	ElCurrentL3Base			: ARRAY[1..2] OF ARRAY[1..100] OF REAL := 
								[
								[0, 0, 0.1, 0.3, 0.45, 0.60, 0.70, 0.80, 0.95, 1.1, 1.3, 1.4, 1.55, 1.6, 1.59,1.55, 
								1.45, 1.3, 1.2, 1.1, 1.05, 1.0, 0.95, 0.9, 0.85, 0.83, 0.80, 0.78, 0.75, 0.74, 0.72,
								0.70, 0.69, 0.69, 0.69, 0.68, 0.68, 0.67, 0.67, 0.65, 0.64, 0.62, 0.60, 0.58, 0.58, 0.57, 0.56, 0.55, 0.55,
								0, 0, 0, 0, 0, 0, 0, 0, 0, 0],
								[0, 0, 0.1, 0.2, 0.3, 0.55, 1.0, 1.3, 1.5, 1.7, 1.8, 1.81, 1.7, 1.5, 1.2, 1.22, 1.19, 1.23,
								1.19, 1.21, 1.18, 1.22, 1.19, 1.23, 1.17, 1.21, 1.20, 1.18, 1.21, 1.18, 1.22, 1.17, 1.23,
								1.19, 1.21, 1.19, 1.20, 1.19, 1.20, 1.19, 1.21, 1.20, 1.20, 1.22, 1.19, 1.21, 1.18, 1.21, 1.2, 1.2,
								1.21, 1.20, 1.20, 1.22, 1.19, 1.21, 1.18, 1.21, 1.2, 1.2]];
END_VAR

IF GVL_Visu.ButtonStart THEN
	
	GVL_Visu.LineRunning := TRUE;
	// simulate motor running signals
	tp1Motor[1](IN:= NOT tp2Motor[1].Q, PT:= T#1S);
	tp2Motor[1](IN:= NOT tp1Motor[1].Q, PT:= T#500MS);
	
	tp1Motor[2](IN:= NOT tp2Motor[2].Q, PT:= T#2S);
	tp2Motor[2](IN:= NOT tp1Motor[2].Q, PT:= T#300MS);
	
	tp1Motor[3](IN:= NOT tp2Motor[3].Q, PT:= T#1.7S);
	tp2Motor[3](IN:= NOT tp1Motor[3].Q, PT:= T#500MS);
	
	tp1Motor[4](IN:= NOT tp2Motor[4].Q, PT:= T#1S);
	tp2Motor[4](IN:= NOT tp1Motor[4].Q, PT:= T#1S);
	
	tp1Motor[5](IN:= NOT tp2Motor[5].Q, PT:= T#500MS);
	tp2Motor[5](IN:= NOT tp1Motor[5].Q, PT:= T#2S);
	
	tp1Motor[6](IN:= NOT tp2Motor[6].Q, PT:= T#1S);
	tp2Motor[6](IN:= NOT tp1Motor[6].Q, PT:= T#300MS);
	
	// simulate auto/manual mode
	tp1AutoMode(IN:= NOT tp2AutoMode.Q, PT:= tp1AutoModeTime);
	tp2AutoMode(IN:= NOT tp1AutoMode.Q, PT:= tp2AutoModeTime);
	
	rtrigAutoMode(CLK:=tp1AutoMode.Q);
	
	// generate random time windows of auto and manual period  
	IF  rtrigAutoMode.Q THEN
		rndTime1 := RDM2(last:=2, low:=0, high:=70);
		tp1AutoModeTime:=T#5S + INT_TO_TIME(rndTime1*100);
		
		rndTime2 := RDM2(last:=5, low:=0, high:=30);
		tp2AutoModeTime:=T#2S + INT_TO_TIME(rndTime2*100);
	END_IF

	GVL_Visu.AutoMode := tp2AutoMode.Q;
	
	
	// simulate vibration sensors
	FOR idx := 1 TO 6 DO
		GVL_Visu.MotorRunning[idx] := tp1Motor[idx].Q;
		
		GVL_Visu.VibrationSensorX[idx] := VibSensorBase[idx] + RDM(0.4);
		GVL_Visu.VibrationSensorY[idx] := VibSensorBase[idx] + RDM(0.2);
		GVL_Visu.VibrationSensorZ[idx] := VibSensorBase[idx] + RDM(0.8);	
	END_FOR
	
	// simulate air supply sensors
	GVL_Visu.AirFlowRate 		:= AirFlowRateBase + 2* RDM(0.5);
	GVL_Visu.AirPressure		:= AirPressureBase + 2 * RDM(0.9); 
	GVL_Visu.AirTemperature		:= AirTemperatureBase + RDM(0.3);
	
	// simulate air valves
	AirValve[1](StartSim			:= TRUE, 
			    ExtendCmdTime		:= T#500MS,
			    ExtendTime 			:= T#1800MS,
			    RetractCmdTime 		:= T#600MS,
			    RetractTime  		:= T#2000MS);
			  
	AirValve[2](StartSim			:= TRUE, 
			    ExtendCmdTime		:= T#50MS,
			    ExtendTime 			:= T#180MS,
			    RetractCmdTime 		:= T#50MS,
			    RetractTime  		:= T#145MS);
				
	AirValve[3](StartSim			:= TRUE, 
			    ExtendCmdTime		:= T#100MS,
			    ExtendTime 			:= T#1200MS,
			    RetractCmdTime 		:= T#120MS,
			    RetractTime  		:= T#1500MS);
				
	AirValve[4](StartSim			:= TRUE, 
			    ExtendCmdTime		:= T#30MS,
			    ExtendTime 			:= T#120MS,
			    RetractCmdTime 		:= T#30MS,
			    RetractTime  		:= T#120MS);
				
	FOR idx := 1 TO 4 DO
		GVL_Visu.AirValve[idx].ExtendCmd := AirValve[idx].ExtendCmd;
		GVL_Visu.AirValve[idx].ExtendFeedback := AirValve[idx].ExtendFeedback;
		GVL_Visu.AirValve[idx].RetractCmd := AirValve[idx].RetractCmd;
		GVL_Visu.AirValve[idx].RetractFeedback := AirValve[idx].RetractFeedback;
		GVL_Visu.AirValvePositionSim[idx] := SEL (NOT GVL_Visu.AirValveEnable[idx], AirValve[idx].nState, 0);
	END_FOR
	
	// simulate product position on the conveyor
	tonProductPos(IN:= NOT tonProductPos.Q, PT:=T#200MS);
	IF tonProductPos.Q THEN
		GVL_Visu.ProductPosition := GVL_Visu.ProductPosition + TO_INT(GVL_Visu.LineSpeed / 5);
	END_IF
	
	IF GVL_Visu.ProductPosition >= 190 THEN
		GVL_Visu.ProductPosition := 0;
	END_IF
	
	// simulate product sensor acitivation
	IF GVL_Visu.ProductPosition >= 175 AND
		 GVL_Visu.ProductPosition <190 THEN
	GVL_Visu.SensorProductActive := TRUE;
	ELSE
		GVL_Visu.SensorProductActive := FALSE;
	END_IF;
	
	// simulate product counting
	rtrigProductSensor(CLK:=GVL_Visu.SensorProductActive);
	IF rtrigProductSensor.Q THEN
		GVL_Visu.OkProductCount := GVL_Visu.OkProductCount + 1;
	END_IF
	
	// simulate electrical current curve of motor 1
	IF GVL_Visu.MotorRunning[1] THEN
		ElecSample1 := ElecSample1+1;
		ElecSample1 := SEL(ElecSample1=60, ElecSample1, 1);
		IF ElecSample1 < 20 OR ElecSample1 > 40 THEN
			ElecCurrentOffsetL1 := RDM(0.67) * 0.05;
			ElecCurrentOffsetL2 := RDM(0.23) * 0.05;
			ElecCurrentOffsetL3 := RDM(0.72) * 0.05;
		ELSE
			ElecCurrentOffsetL1 := RDM(0.31) * 0.05;
			ElecCurrentOffsetL2 := RDM(0.63) * 0.05;
			ElecCurrentOffsetL3 := RDM(0.46) * 0.05;
		END_IF
		GVL_Visu.ElCurrentL1[1] := 	ElCurrentL1Base[1][ElecSample1] + ElecCurrentOffsetL1;
		GVL_Visu.ElCurrentL2[1] := 	ElCurrentL2Base[1][ElecSample1] + ElecCurrentOffsetL2;
		GVL_Visu.ElCurrentL3[1] := 	ElCurrentL3Base[1][ElecSample1] + ElecCurrentOffsetL3;
	ELSE
		ElecSample1 := 0;
		GVL_Visu.ElCurrentL1[1] := 0;
		GVL_Visu.ElCurrentL2[1] := 0;
		GVL_Visu.ElCurrentL3[1] := 0;
	END_IF
	
	// simulate electrical current curve of motor 2
	IF GVL_Visu.MotorRunning[2] THEN
		ElecSample2 := ElecSample2+1;
		ElecSample2 := SEL(ElecSample2=60, ElecSample2, 1);
		GVL_Visu.ElCurrentL1[2] := 	ElCurrentL1Base[2][ElecSample2];
		GVL_Visu.ElCurrentL2[2] := 	ElCurrentL2Base[2][ElecSample2];
		GVL_Visu.ElCurrentL3[2] := 	ElCurrentL3Base[2][ElecSample2];
	ELSE
		ElecSample2 := 0;
		GVL_Visu.ElCurrentL1[2] := 0;
		GVL_Visu.ElCurrentL2[2] := 0;
		GVL_Visu.ElCurrentL3[2] := 0;
	END_IF
	
	// simulate ambient temperature & humidity
	GVL_Visu.AmbientTemperature := 19.0 + 2* RDM(0.7);
	GVL_Visu.AmbientHumidity	:= 60.0 + 3 * RDM(0.5);
	
	// simulate pressure difference for oil contamination sensor
	GVL_Visu.OilDiffPressure := 0.2 + RDM(0.1) * 0.2;
  

ELSE
	GVL_Visu.LineRunning := FALSE;
	tp1AutoMode(IN:=FALSE);
	tp2AutoMode(IN:=FALSE);
	
	GVL_Visu.AutoMode := tp1AutoMode.Q;
	
	FOR idx := 1 TO 4 DO
		AirValve[idx](StartSim := FALSE);
	END_FOR
	
	FOR idx := 1 TO 6 DO
		tp1Motor[idx](IN:= FALSE);
		tp2Motor[idx](IN:= FALSE);	
		GVL_Visu.MotorRunning[idx] := tp1Motor[idx].Q;		
	END_FOR
	
	GVL_Visu.ElCurrentL1[1] := 0;
	GVL_Visu.ElCurrentL2[1] := 0;
	GVL_Visu.ElCurrentL3[1] := 0;
	
	GVL_Visu.ElCurrentL1[2] := 0;
	GVL_Visu.ElCurrentL2[2] := 0;
	GVL_Visu.ElCurrentL3[2] := 0;
	
END_IF

END_PROGRAM

// ---- POUs/PRG_10ms/PRG_03_VibrationAnalytics.TcPOU
PROGRAM PRG_03_VibrationAnalytics
VAR
	VibSensor					: ARRAY [1..6] OF VibrationSensor;
	VibSensorPublishMqtt		: ARRAY [1..6] OF PublishJsonMqtt;	
END_VAR


// PAGE Vibration Sensor 1 ----
VibSensor[1](
    LineName := GVL_const.LineName,
    MachineName := GVL_const.MachineName,
    SensorName := GVL_const.VibSensor1,
    TimeStamp := GVL_SW.Unix_TimeStamp,
    VibAccelX := GVL_Visu.VibrationSensorX[1],
    VibAccelY := GVL_Visu.VibrationSensorY[1],
    VibAccelZ := GVL_Visu.VibrationSensorZ[1],
    SensorTemperature := GVL_SW.VibSensor1Temp,
    MotorState := GVL_Visu.MotorRunning[1],
    Enable := GVL_Visu.LineRunning AND GVL_Visu.VibrationSensorsEnable); // VibrationSensor
VibSensorPublishMqtt[1](
    HostAddress := GVL_const.MqttBrokerIPAddress,
    HostPort := GVL_const.MqttHostPort,
    UserName := GVL_const.MqttUserName,
    UserPassword := GVL_const.MqttPassword,
    JsonPayload := VibSensor[1].MqttJsonPayload,
    PublishCommand := VibSensor[1].PublishMQTT,
    MqttTopic := VibSensor[1].MqttTopic); // PublishJsonMqtt

// PAGE Vibration Sensor 2 ---
VibSensor[2](
    LineName := GVL_const.LineName,
    MachineName := GVL_const.MachineName,
    SensorName := GVL_const.VibSensor2,
    TimeStamp := GVL_SW.Unix_TimeStamp,
    VibAccelX := GVL_Visu.VibrationSensorX[2],
    VibAccelY := GVL_Visu.VibrationSensorY[2],
    VibAccelZ := GVL_Visu.VibrationSensorZ[2],
    SensorTemperature := GVL_SW.VibSensor2Temp,
    MotorState := GVL_Visu.MotorRunning[2],
    Enable := GVL_Visu.LineRunning AND GVL_Visu.VibrationSensorsEnable); // VibrationSensor
VibSensorPublishMqtt[2](
    HostAddress := GVL_const.MqttBrokerIPAddress,
    HostPort := GVL_const.MqttHostPort,
    UserName := GVL_const.MqttUserName,
    UserPassword := GVL_const.MqttPassword,
    JsonPayload := VibSensor[2].MqttJsonPayload,
    PublishCommand := VibSensor[2].PublishMQTT,
    MqttTopic := VibSensor[2].MqttTopic); // PublishJsonMqtt

// PAGE Vibration Sensor 3 ---
VibSensor[3](
    LineName := GVL_const.LineName,
    MachineName := GVL_const.MachineName,
    SensorName := GVL_const.VibSensor3,
    TimeStamp := GVL_SW.Unix_TimeStamp,
    VibAccelX := GVL_Visu.VibrationSensorX[3],
    VibAccelY := GVL_Visu.VibrationSensorY[3],
    VibAccelZ := GVL_Visu.VibrationSensorZ[3],
    SensorTemperature := GVL_SW.VibSensor3Temp,
    MotorState := GVL_Visu.MotorRunning[3],
    Enable := GVL_Visu.LineRunning AND GVL_Visu.VibrationSensorsEnable); // VibrationSensor
VibSensorPublishMqtt[3](
    HostAddress := GVL_const.MqttBrokerIPAddress,
    HostPort := GVL_const.MqttHostPort,
    UserName := GVL_const.MqttUserName,
    UserPassword := GVL_const.MqttPassword,
    JsonPayload := VibSensor[3].MqttJsonPayload,
    PublishCommand := VibSensor[3].PublishMQTT,
    MqttTopic := VibSensor[3].MqttTopic); // PublishJsonMqtt

// PAGE Vibration Sensor 4 ---
VibSensor[4](
    LineName := GVL_const.LineName,
    MachineName := GVL_const.MachineName,
    SensorName := GVL_const.VibSensor4,
    TimeStamp := GVL_SW.Unix_TimeStamp,
    VibAccelX := GVL_Visu.VibrationSensorX[4],
    VibAccelY := GVL_Visu.VibrationSensorY[4],
    VibAccelZ := GVL_Visu.VibrationSensorZ[4],
    SensorTemperature := GVL_SW.VibSensor4Temp,
    MotorState := GVL_Visu.MotorRunning[4],
    Enable := GVL_Visu.LineRunning AND GVL_Visu.VibrationSensorsEnable); // VibrationSensor
VibSensorPublishMqtt[4](
    HostAddress := GVL_const.MqttBrokerIPAddress,
    HostPort := GVL_const.MqttHostPort,
    UserName := GVL_const.MqttUserName,
    UserPassword := GVL_const.MqttPassword,
    JsonPayload := VibSensor[4].MqttJsonPayload,
    PublishCommand := VibSensor[4].PublishMQTT,
    MqttTopic := VibSensor[4].MqttTopic); // PublishJsonMqtt

// PAGE Vibration Sensor 5 ---
VibSensor[5](
    LineName := GVL_const.LineName,
    MachineName := GVL_const.MachineName,
    SensorName := GVL_const.VibSensor5,
    TimeStamp := GVL_SW.Unix_TimeStamp,
    VibAccelX := GVL_Visu.VibrationSensorX[5],
    VibAccelY := GVL_Visu.VibrationSensorY[5],
    VibAccelZ := GVL_Visu.VibrationSensorZ[5],
    SensorTemperature := GVL_SW.VibSensor5Temp,
    MotorState := GVL_Visu.MotorRunning[5],
    Enable := GVL_Visu.LineRunning AND GVL_Visu.VibrationSensorsEnable); // VibrationSensor
VibSensorPublishMqtt[5](
    HostAddress := GVL_const.MqttBrokerIPAddress,
    HostPort := GVL_const.MqttHostPort,
    UserName := GVL_const.MqttUserName,
    UserPassword := GVL_const.MqttPassword,
    JsonPayload := VibSensor[5].MqttJsonPayload,
    PublishCommand := VibSensor[5].PublishMQTT,
    MqttTopic := VibSensor[5].MqttTopic); // PublishJsonMqtt

// PAGE Vibration Sensor 6 ---
VibSensor[6](
    LineName := GVL_const.LineName,
    MachineName := GVL_const.MachineName,
    SensorName := GVL_const.VibSensor6,
    TimeStamp := GVL_SW.Unix_TimeStamp,
    VibAccelX := GVL_Visu.VibrationSensorX[6],
    VibAccelY := GVL_Visu.VibrationSensorY[6],
    VibAccelZ := GVL_Visu.VibrationSensorZ[6],
    SensorTemperature := GVL_SW.VibSensor6Temp,
    MotorState := GVL_Visu.MotorRunning[6],
    Enable := GVL_Visu.LineRunning AND GVL_Visu.VibrationSensorsEnable); // VibrationSensor
VibSensorPublishMqtt[6](
    HostAddress := GVL_const.MqttBrokerIPAddress,
    HostPort := GVL_const.MqttHostPort,
    UserName := GVL_const.MqttUserName,
    UserPassword := GVL_const.MqttPassword,
    JsonPayload := VibSensor[6].MqttJsonPayload,
    PublishCommand := VibSensor[6].PublishMQTT,
    MqttTopic := VibSensor[6].MqttTopic); // PublishJsonMqtt
// GVL.BS1_Accel_RMS_X: input not connected
// GVL.BS1_Accel_RMS_Y: input not connected
// GVL.BS1_Accel_RMS_Z: input not connected
// GVL.Drv_RotTable_25N0_M10_RUNNING: input not connected
// GVL.AutoMode: input not connected
// GVL.BS2_Accel_RMS_X: input not connected
// GVL.BS2_Accel_RMS_Y: input not connected
// GVL.BS2_Accel_RMS_Z: input not connected
// GVL.Drv_RotTable_25N0_M10_RUNNING: input not connected
// GVL.AutoMode: input not connected
// GVL.BS3_Accel_RMS_X: input not connected
// GVL.BS3_Accel_RMS_Y: input not connected
// GVL.BS3_Accel_RMS_Z: input not connected
// GVL.Drv_RotTable_25N0_M10_RUNNING: input not connected
// GVL.AutoMode: input not connected
// GVL.BS4_Accel_RMS_X: input not connected
// GVL.BS4_Accel_RMS_Y: input not connected
// GVL.BS4_Accel_RMS_Z: input not connected
// GVL.Drv_RotTable_25N0_M10_RUNNING: input not connected
// GVL.AutoMode: input not connected
// GVL.BS5_Accel_RMS_X: input not connected
// GVL.BS5_Accel_RMS_Y: input not connected
// GVL.BS5_Accel_RMS_Z: input not connected
// GVL.Drv_InfeedBelt2_10N31_M21_RIGHT_RUNNING: input not connected
// GVL.AutoMode: input not connected
// GVL.BS6_Accel_RMS_X: input not connected
// GVL.BS6_Accel_RMS_Y: input not connected
// GVL.BS6_Accel_RMS_Z: input not connected
// GVL.Drv_InfeedBelt2_10N31_M21_RIGHT_RUNNING: input not connected
// GVL.AutoMode: input not connected

END_PROGRAM

// ---- POUs/PRG_10ms/PRG_07_LineState.TcPOU
PROGRAM PRG_07_LineState
VAR
	CheckLine1Producing: CheckLineProducing;
	
	ValueChangeDetector	:	ARRAY[1..6] OF ValueChangeDetector;
	GenericState		:	ARRAY[1..6] OF GenericState;
	PublishJsonMqtt		:	ARRAY[1..6] OF PublishJsonMqtt;
	tpValueChangeDelay	:	ARRAY[1..6] OF TP;
	
END_VAR


// PAGE Check if line is producing --
CheckLine1Producing(OkProductNumber := GVL_Visu.OkProductCount); // CheckLineProducing
GVL_Visu.LineProducing := CheckLine1Producing.LineProducing;

// PAGE Send line states over MQTT ---
ValueChangeDetector[1](Value := BOOL_TO_INT(GVL_Visu.AutoMode)); // ValueChangeDetector
tpValueChangeDelay[1](IN := ValueChangeDetector[1].ValueChanged, PT := T#50MS); // TP
GenericState[1](
    LineName := GVL_const.LineName,
    MachineName := GVL_const.MachineName,
    StateName := 'AutoMode',
    TimeStamp := GVL_SW.Unix_TimeStamp,
    Value := BOOL_TO_INT(GVL_Visu.AutoMode),
    Enable := tpValueChangeDelay[1].Q); // GenericState
PublishJsonMqtt[1](
    HostAddress := GVL_const.MqttBrokerIPAddress,
    HostPort := GVL_const.MqttHostPort,
    UserName := GVL_const.MqttUserName,
    UserPassword := GVL_const.MqttPassword,
    MqttTopic := GenericState[1].MqttTopic,
    JsonPayload := GenericState[1].MqttJsonPayload,
    PublishCommand := GenericState[1].PublishMQTT); // PublishJsonMqtt
ValueChangeDetector[2](Value := BOOL_TO_INT(GVL_Visu.AutoMode)); // ValueChangeDetector
tpValueChangeDelay[2](IN := ValueChangeDetector[2].ValueChanged, PT := T#50MS); // TP
GenericState[2](
    LineName := GVL_const.LineName,
    MachineName := GVL_const.MachineName,
    StateName := 'DoorOpened',
    TimeStamp := GVL_SW.Unix_TimeStamp,
    Value := BOOL_TO_INT(GVL_Visu.AutoMode),
    Enable := tpValueChangeDelay[2].Q); // GenericState
PublishJsonMqtt[2](
    HostAddress := GVL_const.MqttBrokerIPAddress,
    HostPort := GVL_const.MqttHostPort,
    UserName := GVL_const.MqttUserName,
    UserPassword := GVL_const.MqttPassword,
    MqttTopic := GenericState[2].MqttTopic,
    JsonPayload := GenericState[2].MqttJsonPayload,
    PublishCommand := GenericState[2].PublishMQTT); // PublishJsonMqtt
ValueChangeDetector[3](Value := BOOL_TO_INT(GVL_Visu.LineProducing)); // ValueChangeDetector
tpValueChangeDelay[3](IN := ValueChangeDetector[3].ValueChanged, PT := T#50MS); // TP
GenericState[3](
    LineName := GVL_const.LineName,
    MachineName := GVL_const.MachineName,
    StateName := 'LineProducing',
    TimeStamp := GVL_SW.Unix_TimeStamp,
    Value := BOOL_TO_INT(GVL_Visu.LineProducing),
    Enable := tpValueChangeDelay[3].Q); // GenericState
PublishJsonMqtt[3](
    HostAddress := GVL_const.MqttBrokerIPAddress,
    HostPort := GVL_const.MqttHostPort,
    UserName := GVL_const.MqttUserName,
    UserPassword := GVL_const.MqttPassword,
    MqttTopic := GenericState[3].MqttTopic,
    JsonPayload := GenericState[3].MqttJsonPayload,
    PublishCommand := GenericState[3].PublishMQTT); // PublishJsonMqtt
ValueChangeDetector[4](Value := UINT_TO_INT(GVL_Visu.OkProductCount)); // ValueChangeDetector

END_PROGRAM

// ---- POUs/PRG_10ms/PRG_08_ProductionStatistics.TcPOU
PROGRAM PRG_08_ProductionStatistics
VAR
	PartsPerMinInstant					: PartsPerMinInstant2;
	PartsPerMin							: GenericState;
	PartsPerMinPublishMqtt				: PublishJsonMqtt;
	OkPartsPerMinHistorical				: PartsPerMinHistorical;
END_VAR

PartsPerMinInstant(TotalCount := GVL_Visu.OkProductCount); // PartsPerMinInstant2
GVL_Visu.OkPartsPerMinRate := PartsPerMinInstant.PPM;
PartsPerMin(
    LineName := GVL_const.LineName,
    MachineName := GVL_const.MachineName,
    StateName := 'PartsPerMinute',
    TimeStamp := GVL_SW.Unix_TimeStamp,
    Value := TO_INT(PartsPerMinInstant.PPM),
    Enable := GVL_Visu.LineRunning); // GenericState
PartsPerMinPublishMqtt(
    HostAddress := GVL_const.MqttBrokerIPAddress,
    HostPort := GVL_const.MqttHostPort,
    UserName := GVL_const.MqttUserName,
    UserPassword := GVL_const.MqttPassword,
    MqttTopic := PartsPerMin.MqttTopic,
    JsonPayload := PartsPerMin.MqttJsonPayload,
    PublishCommand := PartsPerMin.PublishMQTT); // PublishJsonMqtt
OkPartsPerMinHistorical(ProductSensor := GVL_Visu.SensorProductActive, PartsPerMinHist := GVL_Visu.OkPartsPerMinHistorical); // PartsPerMinHistorical

END_PROGRAM

// ---- POUs/PRG_10ms/PRG_09_PlcDiagnostic.TcPOU
PROGRAM PRG_09_PlcDiagnostic
VAR
	NetID						: 	STRING := '192.168.1.145.1.1';
	tonRecycle50ms				: 	TON;
	tonRecyclePublishMqtt		: 	TON;
	
	CpuMemoryUsage				:	ReadMemoryUsage;
	CpuUsageEx_Core2			:	TC_CPuUsageEx;
	CpuUsageEx_Core3			:	TC_CPuUsageEx;
	CpuLatencyEx_Core2			:	TC_SysLatencyEx;
	CpuLatencyEx_Core3			:	TC_SysLatencyEx;
	
	PlcDiagState				:	ARRAY [1..5] OF GenericState;
	PlcDiagStatePublishMqtt		:	ARRAY [1..5] OF PublishJsonMqtt;
END_VAR


// PAGE Recycle Timers for general usage ---
tonRecyclePublishMqtt(IN := NOT tonRecyclePublishMqtt.Q, PT := T#2s); // TON
tonRecycle50ms(IN := NOT tonRecycle50ms.Q, PT := T#50ms); // TON

// PAGE PLC Memory usage ---
CpuMemoryUsage(NetID := NetID); // ReadMemoryUsage
PlcDiagState[1](
    LineName := GVL_const.LineName,
    MachineName := GVL_const.MachineName,
    StateName := GVL_const.PlcCpuMemUsage,
    TimeStamp := GVL_SW.Unix_TimeStamp,
    Value := UINT_TO_INT(CpuMemoryUsage.MemUsage)); // GenericState
PlcDiagStatePublishMqtt[1](
    HostAddress := GVL_const.MqttBrokerIPAddress,
    HostPort := GVL_const.MqttHostPort,
    UserName := GVL_const.MqttUserName,
    UserPassword := GVL_const.MqttPassword,
    MqttTopic := PlcDiagState[1].MqttTopic,
    JsonPayload := PlcDiagState[1].MqttJsonPayload,
    PublishCommand := PlcDiagState[1].PublishMQTT); // PublishJsonMqtt

// PAGE PLC CPU usage ---
CpuUsageEx_Core2(bExecute := tonRecycle50ms.Q, tTimeout := T#5S, sNetId := NetID, nCpuId := 2); // TC_CPuUsageEx
PlcDiagState[2](
    LineName := GVL_const.LineName,
    MachineName := GVL_const.MachineName,
    StateName := GVL_const.PlcCpuCore2Usage,
    TimeStamp := GVL_SW.Unix_TimeStamp,
    Value := UDINT_TO_INT(CpuUsageEx_Core2.nUsage),
    Enable := GVL_Visu.LineRunning AND tonRecyclePublishMqtt.Q); // GenericState
PlcDiagStatePublishMqtt[2](
    HostAddress := GVL_const.MqttBrokerIPAddress,
    HostPort := GVL_const.MqttHostPort,
    UserName := GVL_const.MqttUserName,
    UserPassword := GVL_const.MqttPassword,
    MqttTopic := PlcDiagState[2].MqttTopic,
    JsonPayload := PlcDiagState[2].MqttJsonPayload,
    PublishCommand := PlcDiagState[2].PublishMQTT); // PublishJsonMqtt
CpuUsageEx_Core3(bExecute := tonRecycle50ms.Q, tTimeout := T#5S, sNetId := NetID, nCpuId := 3); // TC_CPuUsageEx
PlcDiagState[3](
    LineName := GVL_const.LineName,
    MachineName := GVL_const.MachineName,
    StateName := GVL_const.PlcCpuCore3Usage,
    TimeStamp := GVL_SW.Unix_TimeStamp,
    Value := UDINT_TO_INT(CpuUsageEx_Core3.nUsage),
    Enable := GVL_Visu.LineRunning AND tonRecyclePublishMqtt.Q); // GenericState
PlcDiagStatePublishMqtt[3](
    HostAddress := GVL_const.MqttBrokerIPAddress,
    HostPort := GVL_const.MqttHostPort,
    UserName := GVL_const.MqttUserName,
    UserPassword := GVL_const.MqttPassword,
    MqttTopic := PlcDiagState[3].MqttTopic,
    JsonPayload := PlcDiagState[3].MqttJsonPayload,
    PublishCommand := PlcDiagState[3].PublishMQTT); // PublishJsonMqtt

// PAGE PLC CPU latency
CpuLatencyEx_Core2(bExecute := tonRecycle50ms.Q, tTimeout := T#5S, sNetId := NetID, nCpuId := 2); // TC_SysLatencyEx
PlcDiagState[4](
    LineName := GVL_const.LineName,
    MachineName := GVL_const.MachineName,
    StateName := GVL_const.PlcCpuCore2Jitter,
    TimeStamp := GVL_SW.Unix_TimeStamp,
    Value := UDINT_TO_INT(CpuLatencyEx_Core2.nActual),
    Enable := GVL_Visu.LineRunning AND tonRecyclePublishMqtt.Q); // GenericState
PlcDiagStatePublishMqtt[4](
    HostAddress := GVL_const.MqttBrokerIPAddress,
    HostPort := GVL_const.MqttHostPort,
    UserName := GVL_const.MqttUserName,
    UserPassword := GVL_const.MqttPassword,
    MqttTopic := PlcDiagState[4].MqttTopic,
    JsonPayload := PlcDiagState[4].MqttJsonPayload,
    PublishCommand := PlcDiagState[4].PublishMQTT); // PublishJsonMqtt
CpuLatencyEx_Core3(bExecute := tonRecycle50ms.Q, tTimeout := T#5S, sNetId := NetID, nCpuId := 3); // TC_SysLatencyEx
PlcDiagState[5](
    LineName := GVL_const.LineName,
    MachineName := GVL_const.MachineName,
    StateName := GVL_const.PlcCpuCore3Jitter,
    TimeStamp := GVL_SW.Unix_TimeStamp,
    Value := UDINT_TO_INT(CpuLatencyEx_Core3.nActual),
    Enable := GVL_Visu.LineRunning AND tonRecyclePublishMqtt.Q); // GenericState
PlcDiagStatePublishMqtt[5](
    HostAddress := GVL_const.MqttBrokerIPAddress,
    HostPort := GVL_const.MqttHostPort,
    UserName := GVL_const.MqttUserName,
    UserPassword := GVL_const.MqttPassword,
    MqttTopic := PlcDiagState[5].MqttTopic,
    JsonPayload := PlcDiagState[5].MqttJsonPayload,
    PublishCommand := PlcDiagState[5].PublishMQTT); // PublishJsonMqtt
// GVL_Visu.LineRunning AND tonRecyclePublishMqtt.Q: input not connected

END_PROGRAM

// ---- POUs/PRG_10ms/PRG_11_AirFlowAnalytics.TcPOU
PROGRAM PRG_11_AirFlowAnalytics
VAR
	AirFlowRateSensor: GenericSensor;
	AirPressureSensor: GenericSensor;
	AirTemperatureSensor: GenericSensor;
	
	AirFlowSensorPublishMqtt: PublishJsonMqtt;
	AirPresSensorPublishMqtt: PublishJsonMqtt;
	AirTempSensorPublishMqtt: PublishJsonMqtt;
END_VAR

AirFlowRateSensor(
    LineName := GVL_const.LineName,
    MachineName := GVL_const.MachineName,
    SensorName := GVL_const.AirFlowSensor,
    TimeStamp := GVL_SW.Unix_TimeStamp,
    Value := GVL_Visu.AirFlowRate,
    Enable := GVL_Visu.LineRunning); // GenericSensor
AirFlowSensorPublishMqtt(
    HostAddress := GVL_const.MqttBrokerIPAddress,
    HostPort := GVL_const.MqttHostPort,
    UserName := GVL_const.MqttUserName,
    UserPassword := GVL_const.MqttPassword,
    MqttTopic := AirFlowRateSensor.MqttTopic,
    JsonPayload := AirFlowRateSensor.MqttJsonPayload,
    PublishCommand := AirFlowRateSensor.PublishMQTT); // PublishJsonMqtt
AirPressureSensor(
    LineName := GVL_const.LineName,
    MachineName := GVL_const.MachineName,
    SensorName := GVL_const.AirPresSensor,
    TimeStamp := GVL_SW.Unix_TimeStamp,
    Value := GVL_Visu.AirPressure,
    Enable := GVL_Visu.LineRunning); // GenericSensor
AirPresSensorPublishMqtt(
    HostAddress := GVL_const.MqttBrokerIPAddress,
    HostPort := GVL_const.MqttHostPort,
    UserName := GVL_const.MqttUserName,
    UserPassword := GVL_const.MqttPassword,
    MqttTopic := AirPressureSensor.MqttTopic,
    JsonPayload := AirPressureSensor.MqttJsonPayload,
    PublishCommand := AirPressureSensor.PublishMQTT); // PublishJsonMqtt
AirTemperatureSensor(
    LineName := GVL_const.LineName,
    MachineName := GVL_const.MachineName,
    SensorName := GVL_const.AirTempSensor,
    TimeStamp := GVL_SW.Unix_TimeStamp,
    Value := GVL_Visu.AirTemperature,
    Enable := GVL_Visu.LineRunning); // GenericSensor
AirTempSensorPublishMqtt(
    HostAddress := GVL_const.MqttBrokerIPAddress,
    HostPort := GVL_const.MqttHostPort,
    UserName := GVL_const.MqttUserName,
    UserPassword := GVL_const.MqttPassword,
    MqttTopic := AirTemperatureSensor.MqttTopic,
    JsonPayload := AirTemperatureSensor.MqttJsonPayload,
    PublishCommand := AirTemperatureSensor.PublishMQTT); // PublishJsonMqtt
// GVL_SW.AirVolumetricFlowRate: input not connected
// GVL_SW.AirPressure: input not connected
// GVL_SW.AirTemperature: input not connected

END_PROGRAM

// ---- POUs/PRG_10ms/PRG_10_TempHumidAnalytics.TcPOU
PROGRAM PRG_10_TempHumidAnalytics
VAR
	TempSensor								: GenericSensor;
	HumiditySensor							: GenericSensor;
	
	TempSensorPublishMqtt					: PublishJsonMqtt;
	HumidSensorPublishMqtt					: PublishJsonMqtt;
END_VAR

TempSensor(
    LineName := GVL_const.LineName,
    MachineName := GVL_const.MachineName,
    SensorName := GVL_const.AmbientTempSensor,
    TimeStamp := GVL_SW.Unix_TimeStamp,
    Value := GVL_Visu.AmbientTemperature,
    Enable := GVL_Visu.LineRunning); // GenericSensor
TempSensorPublishMqtt(
    HostAddress := GVL_const.MqttBrokerIPAddress,
    HostPort := GVL_const.MqttHostPort,
    UserName := GVL_const.MqttUserName,
    UserPassword := GVL_const.MqttPassword,
    MqttTopic := TempSensor.MqttTopic,
    JsonPayload := TempSensor.MqttJsonPayload,
    PublishCommand := TempSensor.PublishMQTT); // PublishJsonMqtt
HumiditySensor(
    LineName := GVL_const.LineName,
    MachineName := GVL_const.MachineName,
    SensorName := GVL_const.AmbientHumiditySensor,
    TimeStamp := GVL_SW.Unix_TimeStamp,
    Value := GVL_Visu.AmbientHumidity,
    Enable := GVL_Visu.LineRunning); // GenericSensor
HumidSensorPublishMqtt(
    HostAddress := GVL_const.MqttBrokerIPAddress,
    HostPort := GVL_const.MqttHostPort,
    UserName := GVL_const.MqttUserName,
    UserPassword := GVL_const.MqttPassword,
    MqttTopic := HumiditySensor.MqttTopic,
    JsonPayload := HumiditySensor.MqttJsonPayload,
    PublishCommand := HumiditySensor.PublishMQTT); // PublishJsonMqtt
// GVL_SW.AmbientTempSensor: input not connected
// GVL_SW.AmbientHumiditySensor: input not connected

END_PROGRAM

// ---- POUs/PRG_10ms/PRG_12_OilContaminationAnalytics.TcPOU
PROGRAM PRG_12_OilContaminationAnalytics
VAR
	OilDiffPressSensor: GenericSensor;
	OilDiffPressSensorPublishMqtt: PublishJsonMqtt;
END_VAR

OilDiffPressSensor(
    LineName := GVL_const.LineName,
    MachineName := GVL_const.MachineName,
    SensorName := GVL_const.DiffPressSensor1,
    TimeStamp := GVL_SW.Unix_TimeStamp,
    Value := GVL_Visu.OilDiffPressure,
    Enable := GVL_Visu.LineRunning); // GenericSensor
OilDiffPressSensorPublishMqtt(
    HostAddress := GVL_const.MqttBrokerIPAddress,
    HostPort := GVL_const.MqttHostPort,
    UserName := GVL_const.MqttUserName,
    UserPassword := GVL_const.MqttPassword,
    MqttTopic := OilDiffPressSensor.MqttTopic,
    JsonPayload := OilDiffPressSensor.MqttJsonPayload,
    PublishCommand := OilDiffPressSensor.PublishMQTT); // PublishJsonMqtt
// GVL_SW.DiffPressSensor: input not connected

END_PROGRAM

// ---- GlobalTextList.TcGTLO
TEXTLIST GlobalTextList
  534 = '%d'
  134 = '5              4             3            2           1          0'
  880 = '5             4              3            2          1         0'
  940 = '5             4             3           2          1         0'
  273 = '5             4          3          2          1         0'
  777 = '5           4             3             2            1             0'
  65 = '5           4             3             2            1           0'
  767 = '5           4             3            2           1          0'
  858 = '5          4          3          2          1             0'
  833 = '5          4          3          2          1           0'
  192 = '5          4          3          2          1          0'
  663 = '5         4         3         2         1         0'
  74 = '5       4       3       2       1       0'
  864 = '5     4     3     2     1     0'
  147 = '5  4  3  2  1  0'
  865 = 'Air Valve'
  780 = 'Air Valves'
  202 = 'Disable'
  249 = 'Door Opened'
  558 = 'Last 5 minutes of production'
  931 = 'Line Running'
  430 = 'Minutes     5     4     3     2     1     0'
  189 = 'Parts Per Minute Historical'
  495 = 'Parts Per Minute: %d'
  227 = 'Porduction Line Simulation'
  254 = 'PPM'
  591 = 'Product Counter: %d'
  599 = 'Product Sensor'
  560 = 'Production Line Simulation'
  735 = 'Start / Stop'
  911 = 'Start/Stop'
  508 = 'Vib Sensors'
END_TEXTLIST

// ---- VISU/Visualization1.TcVIS
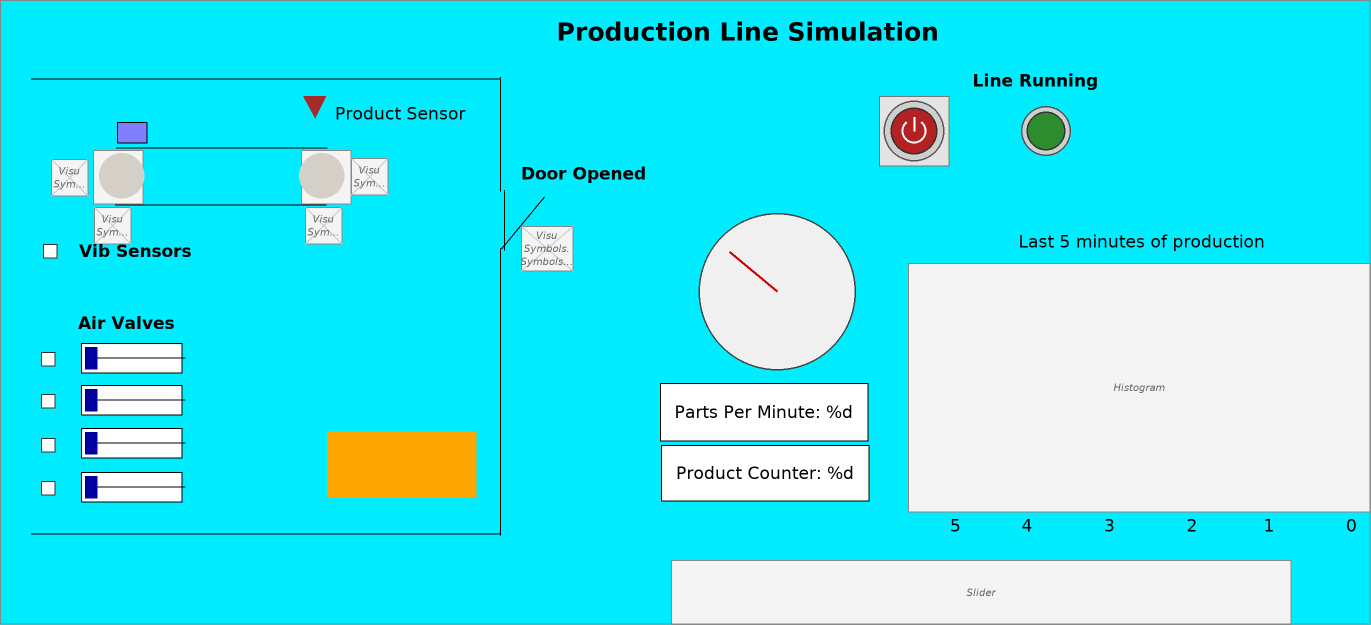
VISUALIZATION Visualization1  // 1371x625
    Pie (93,150 50x54), colour toggle: GVL_Visu.LineRunning
    Line (326,205) (115,205), colour toggle: GVL_Visu.LineRunning
    Line (327,148) (116,148), colour toggle: GVL_Visu.LineRunning
    Pie (301,150 50x54), colour toggle: GVL_Visu.LineRunning
    Meter360 (688,213 178x157), value: GVL_Visu.OkPartsPerMinRate, style: Meter-Meter360-Yellow, scale format: %.1f, scale 0..60
    Lamp1 (1010,102 72x58), variable: GVL_Visu.LineRunning, style: Lamp-Lamp1-Green
    Checkbox (39,344 33x30), variable: GVL_Visu.AirValveEnable[1]
    Line (500,77) (500,191)
    Line (500,248) (500,535)
    Line (500,534) (31,534)
    Line (544,197) (501,249), invisible if: NOT GVL_Visu.AutoMode
    Label (554,9 388x45), "Production Line Simulation"
    Image (521,226 52x45), colour toggle: GVL_Visu.LineRunning, invisible if: NOT GVL_Visu.AutoMode, image: VisuSymbols.Symbols.User
    RoundedRectangle (117,122 30x21)
        p3560616238: GVL_Visu.ProductPosition
    Rectangle (81,343 101x30)
    Group (85,347 100x22)
        p3560616238: GVL_Visu.AirValvePositionSim[1]
        Rectangle (0,0 12x22)
        Line (100,11) (12,11)
    Rectangle (81,385 101x30)
    Group (85,389 100x22)
        p3560616238: GVL_Visu.AirValvePositionSim[2]
        Rectangle (0,0 12x22)
        Line (100,11) (12,11)
    Rectangle (81,428 101x30)
    Group (85,432 100x22)
        p3560616238: GVL_Visu.AirValvePositionSim[3]
        Rectangle (0,0 12x22)
        Line (100,11) (12,11)
    Rectangle (81,472 101x30)
    Group (85,476 100x22)
        p3560616238: GVL_Visu.AirValvePositionSim[4]
        Rectangle (0,0 12x22)
        Line (100,11) (12,11)
    Line (500,79) (31,79)
    PowerSwitch (879,96 70x70), variable: GVL_Visu.ButtonStart, behaviour: TOGGLE, style: Switch-PowerSwitch-Red
    Rectangle (327,431 149x66), colour toggle: GVL_Visu.AutoMode, text list: 'TextList1', text index: GVL_Visu.AutoMode
    Ellipse (99,153 45x45), colour toggle: GVL_Visu.LineRunning
    Slider (671,560 620x65), variable: GVL_Visu.LineSpeed, scale 0..100
    Checkbox (39,386 34x30), variable: GVL_Visu.AirValveEnable[2]
    Checkbox (39,430 34x30), variable: GVL_Visu.AirValveEnable[3]
    Checkbox (39,473 34x30), variable: GVL_Visu.AirValveEnable[4]
    Ellipse (299,153 45x45), colour toggle: GVL_Visu.LineRunning
    Label (513,151 141x45), "Door Opened", invisible if: NOT GVL_Visu.AutoMode
    Polygon (303,96) (315,118) (326,96), colour toggle: GVL_Visu.SensorProductActive
    Label (330,91 141x45), "Product Sensor"
    Label (965,58 141x45), "Line Running"
    Line (504,190) (504,250), invisible if: GVL_Visu.AutoMode
    Label (56,306 141x34), "Air Valves"
    Image (51,159 37x37), angle 90, image: VisuSymbols.Symbols.Marker
    Image (94,207 37x37), image: VisuSymbols.Symbols.Marker
    Image (305,207 37x37), image: VisuSymbols.Symbols.Marker
    Image (351,158 37x37), angle -90, image: VisuSymbols.Symbols.Marker
    Label (65,234 141x34), "Vib Sensors"
    Histogram (908,263 463x249), scale format: %d, scale 0..60
        p1518820177: GVL_Visu.OkPartsPerMinHistorical
        p102497268: GVL_Visu.OkPartsPerMinHistorical
        p788070771: ARRAY [1..5] OF INT
    RoundedRectangle (661,445 208x56), "Product Counter: %d", text variable: GVL_Visu.OkProductCount
    RoundedRectangle (660,383 208x58), "Parts Per Minute: %d", text variable: GVL_Visu.OkPartsPerMinRate
    Label (997,219 290x45), "Last 5 minutes of production"
    Label (947,506 411x39), "5 4 3 2 1 0"
    Checkbox (41,236 33x30), variable: GVL_Visu.VibrationSensorsEnable
END_VISUALIZATION
